(* IEC 61131-3 sources: bcs-engineering-dsl/language/test/generating/array_test/expected, 4 files *)

(* ---- ArrayTestFB_decl.st ---- *)
FUNCTION_BLOCK ArrayTestFB
VAR_INPUT
    iValues: ARRAY [0..9] OF INT;
    iCount: INT;
END_VAR
VAR_OUTPUT
    oSum: INT;
    oAverage: REAL;
    oMaxValue: INT;
    oProcessedValues: ARRAY [0..9] OF INT;
END_VAR
VAR
    i: INT;
    sum: INT := 0;
    maxVal: INT := -32768;
END_VAR

(* ---- ArrayTestFB_impl.st ---- *)
sum := 0;
maxVal := -32768;
FOR i := 0 TO iCount - 1 BY 1 DO
    sum := sum + iValues[i];
    IF iValues[i] > maxVal THEN
        maxVal := iValues[i];
    END_IF;
    oProcessedValues[i] := iValues[i] * 2;
END_FOR;
FOR i := iCount TO 9 DO
    oProcessedValues[i] := 0;
END_FOR;
oSum := sum;
oMaxValue := maxVal;
IF iCount > 0 THEN
    oAverage := sum / iCount;
ELSE
    oAverage := 0;
END_IF;

(* ---- MAIN_decl.st ---- *)
PROGRAM MAIN
VAR
    TestArrays_values: ARRAY [0..9] OF INT := [10, 20, 30, 40, 50, -5, 15, 25, 35, 45];
    TestArrays_count: INT := 8;
    TestArrays_sum: INT;
    TestArrays_average: REAL;
    TestArrays_maxValue: INT;
    TestArrays_processedValues: ARRAY [0..9] OF INT;
    TestArrays_twoDimensionalArray: ARRAY [0..1, 0..2] OF INT := [1, 2, 3, 4, 5, 6];
    TestArrays_rowCount: INT := 2;
    TestArrays_colCount: INT := 3;
    TestArrays_rowSum: ARRAY [0..1] OF INT := [0, 0];
    TestArrays_colSum: ARRAY [0..2] OF INT := [0, 0, 0];
    TestArrayOperations_array1: ARRAY [0..4] OF INT := [1, 2, 3, 4, 5];
    TestArrayOperations_array2: ARRAY [0..4] OF INT := [6, 7, 8, 9, 10];
    TestArrayOperations_resultArray: ARRAY [0..4] OF INT;
    TestArrayOperations_resultArray2: ARRAY [0..4] OF INT;
    i: INT := 0;
    j: INT := 0;
    ArrayTestFBInstance1: ArrayTestFB;
END_VAR

(* ---- MAIN_impl.st ---- *)
// Control Unit 'TestArrays'
ArrayTestFBInstance1(iValues:=TestArrays_values, iCount:=TestArrays_count);
TestArrays_sum := ArrayTestFBInstance1.oSum;
TestArrays_average := ArrayTestFBInstance1.oAverage;
TestArrays_maxValue := ArrayTestFBInstance1.oMaxValue;
TestArrays_processedValues := ArrayTestFBInstance1.oProcessedValues;

FOR i := 0 TO TestArrays_rowCount - 1 DO
    FOR j := 0 TO TestArrays_colCount - 1 DO
        TestArrays_rowSum[i] := TestArrays_rowSum[i] + TestArrays_twoDimensionalArray[i, j];
        TestArrays_colSum[j] := TestArrays_colSum[j] + TestArrays_twoDimensionalArray[i, j];
    END_FOR;
END_FOR;
// Control Unit 'TestArrayOperations'
FOR i := 0 TO 4 DO
    TestArrayOperations_resultArray[i] := TestArrayOperations_array1[i] + TestArrayOperations_array2[i];
END_FOR;
FOR i := 0 TO 4 DO
    TestArrayOperations_resultArray2[i] := TestArrayOperations_array1[i] * TestArrayOperations_array2[i];
END_FOR;
